Staubli VAL3: SplitNumS.pgx

public program SplitNumS(string x_Source, num& x_Res[], string& x_sChar[], bool& x_bRes)
  local num l_nNum
begin

  call SplitString(x_Source,sBuff,x_sChar,x_bRes)
  if !x_bRes
    return
  endIf



  //把分解的字符串转化为数字量
  for l_nNum=0 to min(size(sBuff)-1,size(x_Res)-1)
    toNum(sBuff[l_nNum],x_Res[l_nNum],x_bRes)
    if !x_bRes
      return
    endIf
  endFor




end
